Fanuc KAREL source: kt00908.KL

-- PROVISIONAL review KL for V940-1; original PC SHA256 58e31462c0bec74f2b7e660bbb42c6c02fc5566ae6c6bd362131801a7485ba75
-- Incomplete behavior may be omitted. Consult companion uncertainty JSON. Do not deploy.
PROGRAM KT00908
%NOLOCKGROUP
BEGIN
  -- V9_ZERO_TABLE_METADATA_HINT layout=0002_ascii; no indexed target words; source/name/runtime held
  -- UNRESOLVED_PC offsets 5-28; opcodes 27,22,1C,31,4A
  -- UNRESOLVED_PC offsets 33-37; opcodes 7F
END KT00908
